// TIA Portal V20 export
ORGANIZATION_BLOCK "Main"   // OB1, LAD, ProgramCycle
TITLE = "Main Program Sweep (Cycle)"
// stored: AutoNumber false, IsIECCheckEnabled true, SetENOAutomatically true
   VAR_INPUT
      Initial_Call : Bool;   // Initial call of this OB
      Remanence : Bool;   // =True, if remanent data are available
   END_VAR
   VAR_TEMP   // added for the SCL form of the ladder/FBD networks
      _w1 : Bool;
      _w2 : Bool;
      _w3 : Bool;
      _w4 : Bool;
      _w5 : Bool;
      _w6 : Bool;
   END_VAR
BEGIN

REGION Network 1: First Cycle
   // Set bit to true in first cycle, and false in all other cycles
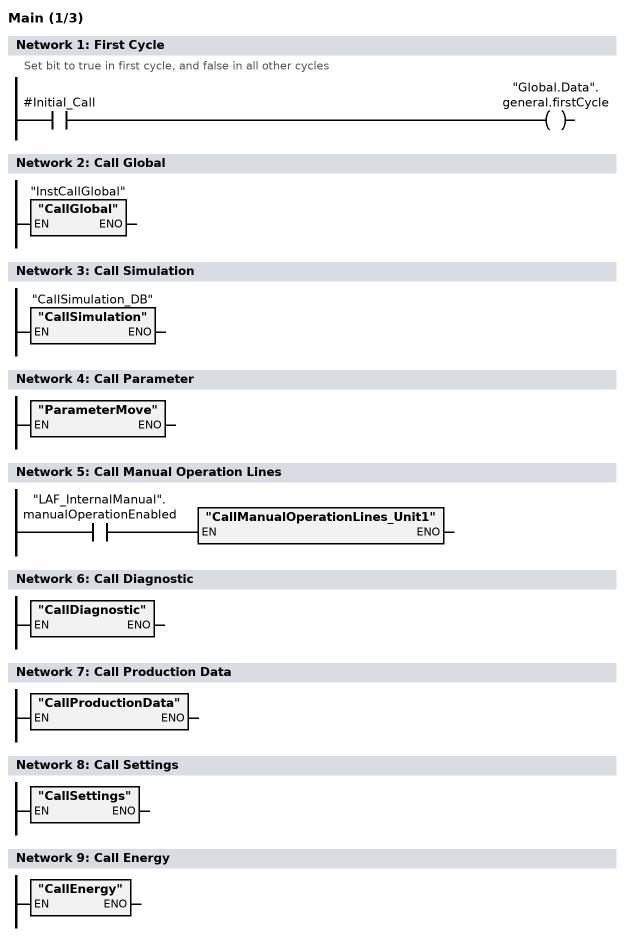
   RUNG wire#powerrail
      Contact( #Initial_Call )
      Coil( "Global.Data".general.firstCycle )
   END_RUNG
   // the same network as SCL:
   "Global.Data".general.firstCycle := #Initial_Call;
END_REGION

REGION Network 2: Call Global
   RUNG wire#powerrail
      "InstCallGlobal"()
   END_RUNG
   // the same network as SCL:
   "InstCallGlobal"();   // "CallGlobal"
END_REGION

REGION Network 3: Call Simulation
   RUNG wire#powerrail
      "CallSimulation_DB"()
   END_RUNG
   // the same network as SCL:
   "CallSimulation_DB"();   // "CallSimulation"
END_REGION

REGION Network 4: Call Parameter
   RUNG wire#powerrail
      "ParameterMove"()
   END_RUNG
   // the same network as SCL:
   "ParameterMove"();
END_REGION

REGION Network 5: Call Manual Operation Lines
   RUNG wire#powerrail
      Contact( "LAF_InternalManual".manualOperationEnabled )
      "CallManualOperationLines_Unit1"()
   END_RUNG
   // the same network as SCL:
   IF "LAF_InternalManual".manualOperationEnabled THEN "CallManualOperationLines_Unit1"(); END_IF;
END_REGION

REGION Network 6: Call Diagnostic
   RUNG wire#powerrail
      "CallDiagnostic"()
   END_RUNG
   // the same network as SCL:
   "CallDiagnostic"();
END_REGION

REGION Network 7: Call Production Data
   RUNG wire#powerrail
      "CallProductionData"()
   END_RUNG
   // the same network as SCL:
   "CallProductionData"();
END_REGION

REGION Network 8: Call Settings
   RUNG wire#powerrail
      "CallSettings"()
   END_RUNG
   // the same network as SCL:
   "CallSettings"();
END_REGION

REGION Network 9: Call Energy
   RUNG wire#powerrail
      "CallEnergy"()
   END_RUNG
   // the same network as SCL:
   "CallEnergy"();
END_REGION

REGION Network 10: HMI SpecialFuction Button Control
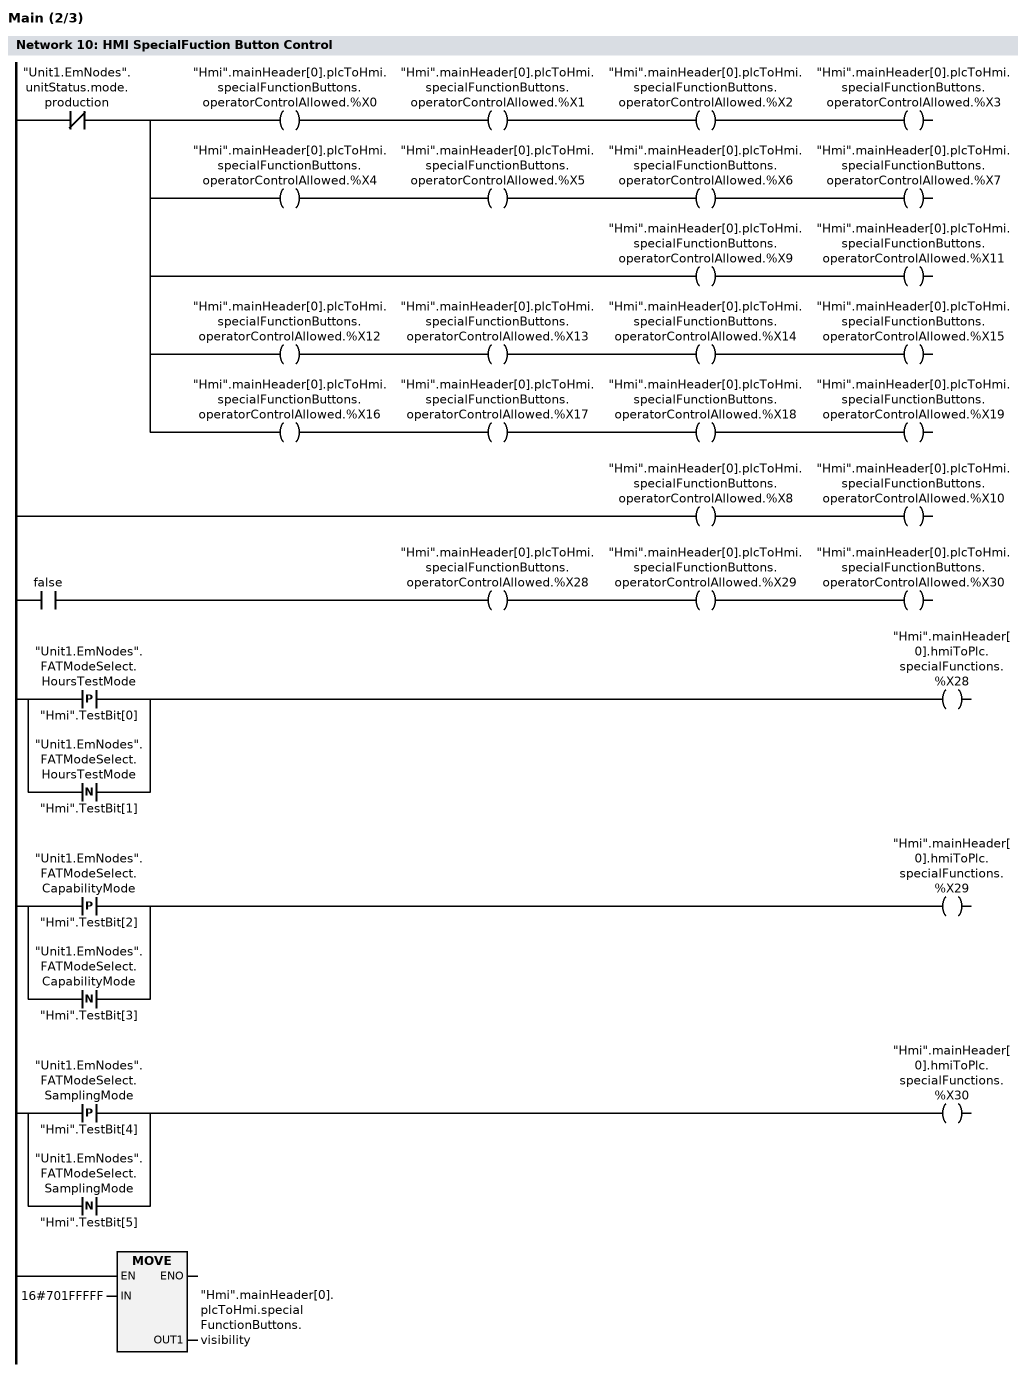
   RUNG wire#powerrail
      I_Contact( "Unit1.EmNodes".unitStatus.mode.production )
      wire#w1
      Coil( "Hmi".mainHeader[0].plcToHmi.specialFunctionButtons.operatorControlAllowed.%X0 )
      Coil( "Hmi".mainHeader[0].plcToHmi.specialFunctionButtons.operatorControlAllowed.%X1 )
      Coil( "Hmi".mainHeader[0].plcToHmi.specialFunctionButtons.operatorControlAllowed.%X2 )
      Coil( "Hmi".mainHeader[0].plcToHmi.specialFunctionButtons.operatorControlAllowed.%X3 )
   END_RUNG
   RUNG wire#w1
      Coil( "Hmi".mainHeader[0].plcToHmi.specialFunctionButtons.operatorControlAllowed.%X4 )
      Coil( "Hmi".mainHeader[0].plcToHmi.specialFunctionButtons.operatorControlAllowed.%X5 )
      Coil( "Hmi".mainHeader[0].plcToHmi.specialFunctionButtons.operatorControlAllowed.%X6 )
      Coil( "Hmi".mainHeader[0].plcToHmi.specialFunctionButtons.operatorControlAllowed.%X7 )
   END_RUNG
   RUNG wire#w1
      Coil( "Hmi".mainHeader[0].plcToHmi.specialFunctionButtons.operatorControlAllowed.%X9 )
      Coil( "Hmi".mainHeader[0].plcToHmi.specialFunctionButtons.operatorControlAllowed.%X11 )
   END_RUNG
   RUNG wire#w1
      Coil( "Hmi".mainHeader[0].plcToHmi.specialFunctionButtons.operatorControlAllowed.%X12 )
      Coil( "Hmi".mainHeader[0].plcToHmi.specialFunctionButtons.operatorControlAllowed.%X13 )
      Coil( "Hmi".mainHeader[0].plcToHmi.specialFunctionButtons.operatorControlAllowed.%X14 )
      Coil( "Hmi".mainHeader[0].plcToHmi.specialFunctionButtons.operatorControlAllowed.%X15 )
   END_RUNG
   RUNG wire#w1
      Coil( "Hmi".mainHeader[0].plcToHmi.specialFunctionButtons.operatorControlAllowed.%X16 )
      Coil( "Hmi".mainHeader[0].plcToHmi.specialFunctionButtons.operatorControlAllowed.%X17 )
      Coil( "Hmi".mainHeader[0].plcToHmi.specialFunctionButtons.operatorControlAllowed.%X18 )
      Coil( "Hmi".mainHeader[0].plcToHmi.specialFunctionButtons.operatorControlAllowed.%X19 )
   END_RUNG
   RUNG wire#powerrail
      Coil( "Hmi".mainHeader[0].plcToHmi.specialFunctionButtons.operatorControlAllowed.%X8 )
      Coil( "Hmi".mainHeader[0].plcToHmi.specialFunctionButtons.operatorControlAllowed.%X10 )
   END_RUNG
   RUNG wire#powerrail
      Contact( false )
      Coil( "Hmi".mainHeader[0].plcToHmi.specialFunctionButtons.operatorControlAllowed.%X28 )
      Coil( "Hmi".mainHeader[0].plcToHmi.specialFunctionButtons.operatorControlAllowed.%X29 )
      Coil( "Hmi".mainHeader[0].plcToHmi.specialFunctionButtons.operatorControlAllowed.%X30 )
   END_RUNG
   RUNG wire#powerrail
      P_Contact(operand := "Unit1.EmNodes".FATModeSelect.HoursTestMode, bit := "Hmi".TestBit[0])
      wire#w2
      Coil( "Hmi".mainHeader[0].hmiToPlc.specialFunctions.%X28 )
   END_RUNG
   RUNG wire#powerrail
      N_Contact(operand := "Unit1.EmNodes".FATModeSelect.HoursTestMode, bit := "Hmi".TestBit[1])
   END_RUNG wire#w2
   RUNG wire#powerrail
      P_Contact(operand := "Unit1.EmNodes".FATModeSelect.CapabilityMode, bit := "Hmi".TestBit[2])
      wire#w3
      Coil( "Hmi".mainHeader[0].hmiToPlc.specialFunctions.%X29 )
   END_RUNG
   RUNG wire#powerrail
      N_Contact(operand := "Unit1.EmNodes".FATModeSelect.CapabilityMode, bit := "Hmi".TestBit[3])
   END_RUNG wire#w3
   RUNG wire#powerrail
      P_Contact(operand := "Unit1.EmNodes".FATModeSelect.SamplingMode, bit := "Hmi".TestBit[4])
      wire#w4
      Coil( "Hmi".mainHeader[0].hmiToPlc.specialFunctions.%X30 )
   END_RUNG
   RUNG wire#powerrail
      N_Contact(operand := "Unit1.EmNodes".FATModeSelect.SamplingMode, bit := "Hmi".TestBit[5])
   END_RUNG wire#w4
   RUNG wire#powerrail
      Move(in := 16#701FFFFF, out1 => "Hmi".mainHeader[0].plcToHmi.specialFunctionButtons.visibility)
   END_RUNG
   // the same network as SCL:
   "Hmi".mainHeader[0].plcToHmi.specialFunctionButtons.operatorControlAllowed.%X0 := NOT "Unit1.EmNodes".unitStatus.mode.production;
   "Hmi".mainHeader[0].plcToHmi.specialFunctionButtons.operatorControlAllowed.%X1 := NOT "Unit1.EmNodes".unitStatus.mode.production;
   "Hmi".mainHeader[0].plcToHmi.specialFunctionButtons.operatorControlAllowed.%X2 := NOT "Unit1.EmNodes".unitStatus.mode.production;
   "Hmi".mainHeader[0].plcToHmi.specialFunctionButtons.operatorControlAllowed.%X3 := NOT "Unit1.EmNodes".unitStatus.mode.production;
   "Hmi".mainHeader[0].plcToHmi.specialFunctionButtons.operatorControlAllowed.%X4 := NOT "Unit1.EmNodes".unitStatus.mode.production;
   "Hmi".mainHeader[0].plcToHmi.specialFunctionButtons.operatorControlAllowed.%X5 := NOT "Unit1.EmNodes".unitStatus.mode.production;
   "Hmi".mainHeader[0].plcToHmi.specialFunctionButtons.operatorControlAllowed.%X6 := NOT "Unit1.EmNodes".unitStatus.mode.production;
   "Hmi".mainHeader[0].plcToHmi.specialFunctionButtons.operatorControlAllowed.%X7 := NOT "Unit1.EmNodes".unitStatus.mode.production;
   "Hmi".mainHeader[0].plcToHmi.specialFunctionButtons.operatorControlAllowed.%X9 := NOT "Unit1.EmNodes".unitStatus.mode.production;
   "Hmi".mainHeader[0].plcToHmi.specialFunctionButtons.operatorControlAllowed.%X11 := NOT "Unit1.EmNodes".unitStatus.mode.production;
   "Hmi".mainHeader[0].plcToHmi.specialFunctionButtons.operatorControlAllowed.%X12 := NOT "Unit1.EmNodes".unitStatus.mode.production;
   "Hmi".mainHeader[0].plcToHmi.specialFunctionButtons.operatorControlAllowed.%X13 := NOT "Unit1.EmNodes".unitStatus.mode.production;
   "Hmi".mainHeader[0].plcToHmi.specialFunctionButtons.operatorControlAllowed.%X14 := NOT "Unit1.EmNodes".unitStatus.mode.production;
   "Hmi".mainHeader[0].plcToHmi.specialFunctionButtons.operatorControlAllowed.%X15 := NOT "Unit1.EmNodes".unitStatus.mode.production;
   "Hmi".mainHeader[0].plcToHmi.specialFunctionButtons.operatorControlAllowed.%X16 := NOT "Unit1.EmNodes".unitStatus.mode.production;
   "Hmi".mainHeader[0].plcToHmi.specialFunctionButtons.operatorControlAllowed.%X17 := NOT "Unit1.EmNodes".unitStatus.mode.production;
   "Hmi".mainHeader[0].plcToHmi.specialFunctionButtons.operatorControlAllowed.%X18 := NOT "Unit1.EmNodes".unitStatus.mode.production;
   "Hmi".mainHeader[0].plcToHmi.specialFunctionButtons.operatorControlAllowed.%X19 := NOT "Unit1.EmNodes".unitStatus.mode.production;
   "Hmi".mainHeader[0].plcToHmi.specialFunctionButtons.operatorControlAllowed.%X8 := TRUE;
   "Hmi".mainHeader[0].plcToHmi.specialFunctionButtons.operatorControlAllowed.%X10 := TRUE;
   "Hmi".mainHeader[0].plcToHmi.specialFunctionButtons.operatorControlAllowed.%X28 := false;
   "Hmi".mainHeader[0].plcToHmi.specialFunctionButtons.operatorControlAllowed.%X29 := false;
   "Hmi".mainHeader[0].plcToHmi.specialFunctionButtons.operatorControlAllowed.%X30 := false;
   #_w1 := "Unit1.EmNodes".FATModeSelect.HoursTestMode AND NOT "Hmi".TestBit[0];   // rising edge of "Unit1.EmNodes".FATModeSelect.HoursTestMode
   "Hmi".TestBit[0] := "Unit1.EmNodes".FATModeSelect.HoursTestMode;
   #_w2 := NOT "Unit1.EmNodes".FATModeSelect.HoursTestMode AND "Hmi".TestBit[1];   // falling edge of "Unit1.EmNodes".FATModeSelect.HoursTestMode
   "Hmi".TestBit[1] := "Unit1.EmNodes".FATModeSelect.HoursTestMode;
   "Hmi".mainHeader[0].hmiToPlc.specialFunctions.%X28 := #_w1 OR #_w2;
   #_w3 := "Unit1.EmNodes".FATModeSelect.CapabilityMode AND NOT "Hmi".TestBit[2];   // rising edge of "Unit1.EmNodes".FATModeSelect.CapabilityMode
   "Hmi".TestBit[2] := "Unit1.EmNodes".FATModeSelect.CapabilityMode;
   #_w4 := NOT "Unit1.EmNodes".FATModeSelect.CapabilityMode AND "Hmi".TestBit[3];   // falling edge of "Unit1.EmNodes".FATModeSelect.CapabilityMode
   "Hmi".TestBit[3] := "Unit1.EmNodes".FATModeSelect.CapabilityMode;
   "Hmi".mainHeader[0].hmiToPlc.specialFunctions.%X29 := #_w3 OR #_w4;
   #_w5 := "Unit1.EmNodes".FATModeSelect.SamplingMode AND NOT "Hmi".TestBit[4];   // rising edge of "Unit1.EmNodes".FATModeSelect.SamplingMode
   "Hmi".TestBit[4] := "Unit1.EmNodes".FATModeSelect.SamplingMode;
   #_w6 := NOT "Unit1.EmNodes".FATModeSelect.SamplingMode AND "Hmi".TestBit[5];   // falling edge of "Unit1.EmNodes".FATModeSelect.SamplingMode
   "Hmi".TestBit[5] := "Unit1.EmNodes".FATModeSelect.SamplingMode;
   "Hmi".mainHeader[0].hmiToPlc.specialFunctions.%X30 := #_w5 OR #_w6;
   "Hmi".mainHeader[0].plcToHmi.specialFunctionButtons.visibility := 16#701FFFFF;
END_REGION

REGION Network 11
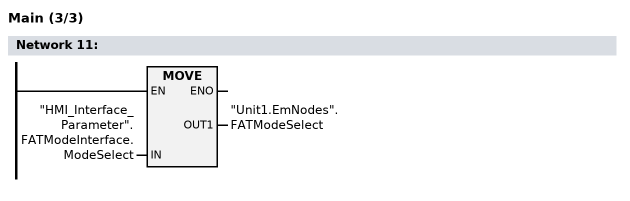
   RUNG wire#powerrail
      Move(in := "HMI_Interface_Parameter".FATModeInterface.ModeSelect, out1 => "Unit1.EmNodes".FATModeSelect)
   END_RUNG
   // the same network as SCL:
   "Unit1.EmNodes".FATModeSelect := "HMI_Interface_Parameter".FATModeInterface.ModeSelect;
END_REGION
END_ORGANIZATION_BLOCK
